Fanuc TP program (LS listing): FIINIT.LS

/PROG  FIINIT
/ATTR
OWNER		= MNEDITOR;
COMMENT		= "FiInit";
PROG_SIZE	= 0;
CREATE		= DATE 26-01-01  TIME 00:00:00;
MODIFIED	= DATE 26-01-01  TIME 00:00:00;
FILE_NAME	= ;
VERSION		= 0;
LINE_COUNT	= 106;
MEMORY_SIZE	= 0;
PROTECT		= READ_WRITE;
TCD:  STACK_SIZE	= 0,
      TASK_PRIORITY	= 50,
      TIME_SLICE	= 0,
      BUSY_LAMP_OFF	= 0,
      ABORT_REQUEST	= 0,
      PAUSE_REQUEST	= 0;
DEFAULT_GROUP	= 1,*,*,*,*;
CONTROL_CODE	= 00000000 00000000;
/MN
   1:  !CrossArm EVALUATION copy ;
   2:  !production use needs a licence ;
   3:  !RAPID FuncInlineProbe.FiInit ;
   4:  !l.133 fiT1:=MakeTool(fiGrip,fiOf ;
   5:  !l.133 fiT1.tframe:=PoseMult(fiGr ;
   6:  PR[84]=PR[98]    ;
   7:  PR[84,2]=PR[84,2]+25    ;
   8:  PR[84,3]=PR[84,3]+40    ;
   9:  PR[84,4]=0    ;
  10:  PR[84,5]=0    ;
  11:  PR[84,6]=0    ;
  12:  UTOOL[1]=PR[84] ;
  13:  !l.134 fiT2:=MakeTool(fiGrip,fiOf ;
  14:  !l.134 fiT2.tframe:=PoseMult(fiGr ;
  15:  PR[84]=PR[98]    ;
  16:  PR[84,2]=PR[84,2]-25    ;
  17:  PR[84,3]=PR[84,3]+40    ;
  18:  PR[84,4]=0    ;
  19:  PR[84,5]=0    ;
  20:  PR[84,6]=0    ;
  21:  UTOOL[3]=PR[84] ;
  22:  !l.135 fiT3:=MakeTool(fiGrip,fiOf ;
  23:  !l.135 fiT3.tframe:=PoseMult(fiGr ;
  24:  PR[84]=PR[98]    ;
  25:  PR[84,1]=PR[84,1]+30    ;
  26:  PR[84,3]=PR[84,3]+62    ;
  27:  PR[84,4]=30    ;
  28:  PR[84,5]=0    ;
  29:  PR[84,6]=0    ;
  30:  UTOOL[4]=PR[84] ;
  31:  !l.136 fiT4:=MakeTool(fiGrip,fiOf ;
  32:  !l.136 fiT4.tframe:=PoseMult(fiGr ;
  33:  PR[84]=PR[98]    ;
  34:  PR[84,1]=PR[84,1]+20    ;
  35:  PR[84,3]=PR[84,3]+30    ;
  36:  PR[84,4]=0    ;
  37:  PR[84,5]=45    ;
  38:  PR[84,6]=0    ;
  39:  UTOOL[5]=PR[84] ;
  40:  !l.137 fiHeavy:=WithLoad(fiGrip,6 ;
  41:  !l.137 fiHeavy.tframe:=fiGrip.tfr ;
  42:  PR[84]=PR[98]    ;
  43:  UTOOL[6]=PR[84] ;
  44:  !l.138 fiShift:=Shifted(fiGrip,25 ;
  45:  !l.138 fiShift.tframe:=fiGrip.tfr ;
  46:  PR[84]=PR[98]    ;
  47:  UTOOL[7]=PR[84] ;
  48:  !l.138 fiShift.tframe.trans.z:=fi ;
  49:  PR[84]=UTOOL[7] ;
  50:  PR[84,3]=PR[84,3]+25    ;
  51:  UTOOL[7]=PR[84] ;
  52:  !l.139 fiT5:=MakeTool(fiCam,fiOfs ;
  53:  !l.139 fiT5.tframe:=PoseMult(fiCa ;
  54:  PR[80]=PR[97]    ;
  55:  PR[79,1]=0    ;
  56:  PR[79,2]=0    ;
  57:  PR[79,3]=35    ;
  58:  PR[79,4]=0    ;
  59:  PR[79,5]=0    ;
  60:  PR[79,6]=0    ;
  61:  CALL CA_POSEMULT(80,79,84) ;
  62:  UTOOL[8]=PR[84] ;
  63:  !l.140 fiT6:=MakeTool(fiCam,fiOfs ;
  64:  !l.140 fiT6.tframe:=PoseMult(fiCa ;
  65:  PR[80]=PR[97]    ;
  66:  PR[79,1]=15    ;
  67:  PR[79,2]=0    ;
  68:  PR[79,3]=20    ;
  69:  PR[79,4]=0    ;
  70:  PR[79,5]=0    ;
  71:  PR[79,6]=(-40)    ;
  72:  CALL CA_POSEMULT(80,79,84) ;
  73:  UTOOL[9]=PR[84] ;
  74:  !l.141 fiTurn:=TurnTool(fiCam,-30 ;
  75:  !l.141 fiTurn.tframe:=PoseMult(fi ;
  76:  PR[80]=PR[97]    ;
  77:  PR[79,1]=0    ;
  78:  PR[79,2]=0    ;
  79:  PR[79,3]=0    ;
  80:  PR[79,4]=0    ;
  81:  PR[79,5]=0    ;
  82:  PR[79,6]=(-30)    ;
  83:  CALL CA_POSEMULT(80,79,84) ;
  84:  PR[99]=PR[84]    ;
  85:  !l.142 fiLeft:=ShiftFixture(fiTab ;
  86:  !l.142 fiLeft.uframe:=PoseMult(fi ;
  87:  PR[80]=UFRAME[3] ;
  88:  PR[79,1]=0    ;
  89:  PR[79,2]=(-150)    ;
  90:  PR[79,3]=0    ;
  91:  PR[79,4]=0    ;
  92:  PR[79,5]=0    ;
  93:  PR[79,6]=0    ;
  94:  CALL CA_POSEMULT(80,79,84) ;
  95:  UFRAME[1]=PR[84] ;
  96:  !l.143 fiRight:=ShiftFixture(fiTa ;
  97:  !l.143 fiRight.uframe:=PoseMult(f ;
  98:  PR[80]=UFRAME[3] ;
  99:  PR[79,1]=0    ;
 100:  PR[79,2]=150    ;
 101:  PR[79,3]=0    ;
 102:  PR[79,4]=0    ;
 103:  PR[79,5]=0    ;
 104:  PR[79,6]=10    ;
 105:  CALL CA_POSEMULT(80,79,84) ;
 106:  UFRAME[2]=PR[84] ;
/POS
/END
